KUKA KRL program: Comm010Config.src, Comm010Config.dat

--- Comm010Config.src ---
&ACCESS RVO1
&COMMENT Comm010 Config
&PARAM EDITMASK = *
&PARAM TEMPLATE = C:\KRC\Roboter\Template\vorgabe
&PARAM DISKPATH = KRC:\R1\Program\SbtComm010Stack
DEF Comm010Config( )
;FOLD INI;%{PE}
  ;FOLD BASISTECH INI
    GLOBAL INTERRUPT DECL 3 WHEN $STOPMESS==TRUE DO IR_STOPM ( )
    INTERRUPT ON 3
    BAS (#INITMOV,0 )
  ;ENDFOLD (BASISTECH INI)
  ;FOLD USER INI
    ;Make your modifications here

  ;ENDFOLD (USER INI)
;ENDFOLD (INI)
;FOLD Basic.SetBusCommTimeout IN Timeout: -1 ms ;%{PE}
BusTimeout = -1
;ENDFOLD
;FOLD SbtComm010.FsConfig IN Fs Id: 1, IN Max: Max1, IN Min: Min1 ;%{PE}
Comm010LimUp[1] = Max1
Comm010LimDown[1] = Min1
;ENDFOLD
;FOLD SbtComm010.FsConfig IN Fs Id: 2, IN Max: Max2, IN Min: Min2 ;%{PE}
Comm010LimUp[2] = Max2
Comm010LimDown[2] = Min2
;ENDFOLD
;FOLD SbtComm010.FsConfig IN Fs Id: 3, IN Max: Max3, IN Min: Min3 ;%{PE}
Comm010LimUp[3] = Max3
Comm010LimDown[3] = Min3
;ENDFOLD
;FOLD SbtComm010.FsConfig IN Fs Id: 4, IN Max: Max4, IN Min: Min4 ;%{PE}
Comm010LimUp[4] = Max4
Comm010LimDown[4] = Min4
;ENDFOLD
;FOLD SbtComm010.FsConfig IN Fs Id: 5, IN Max: Max5, IN Min: Min5 ;%{PE}
Comm010LimUp[5] = Max5
Comm010LimDown[5] = Min5
;ENDFOLD
;FOLD SbtComm010.FsConfig IN Fs Id: 6, IN Max: Max6, IN Min: Min6 ;%{PE}
Comm010LimUp[6] = Max6
Comm010LimDown[6] = Min6
;ENDFOLD
;FOLD SbtComm010.FsConfig IN Fs Id: 7, IN Max: Max7, IN Min: Min7 ;%{PE}
Comm010LimUp[7] = Max7
Comm010LimDown[7] = Min7
;ENDFOLD
;FOLD SbtComm010.FsConfig IN Fs Id: 8, IN Max: Max8, IN Min: Min8 ;%{PE}
Comm010LimUp[8] = Max8
Comm010LimDown[8] = Min8
;ENDFOLD


END

--- Comm010Config.dat ---
&ACCESS RVO1
&PARAM EDITMASK = *
&PARAM TEMPLATE = C:\KRC\Roboter\Template\vorgabe
&PARAM DISKPATH = KRC:\R1\Program\SbtComm010Stack
DEFDAT Comm010Config
;FOLD EXTERNAL DECLARATIONS;%{PE}%MKUKATPBASIS,%CEXT,%VCOMMON,%P
;FOLD BASISTECH EXT;%{PE}%MKUKATPBASIS,%CEXT,%VEXT,%P
EXT  BAS (BAS_COMMAND  :IN,REAL  :IN )
DECL INT SUCCESS
;ENDFOLD (BASISTECH EXT)
;FOLD USER EXT;%{E}%MKUKATPUSER,%CEXT,%VEXT,%P
;Make your modifications here

;ENDFOLD (USER EXT)
;ENDFOLD (EXTERNAL DECLARATIONS)
DECL vector_t Max1={X 3000.00,Y 3000.00,Z 3000.00}
DECL vector_t Min1={X -3000.00,Y -3000.00,Z -3000.00}
DECL MODULEPARAM_T LAST_TP_PARAMS={PARAMS[] "SBTCOMM010.FSID=8; SBTCOMM010.MAX=Max8; SBTCOMM010.MIN=Min8; BASIC.TIMEOUT=-1    "}
DECL vector_t Max2={X 3000.00,Y 3000.00,Z 3000.00}
DECL vector_t Min2={X -3000.00,Y -3000.00,Z -3000.00}
DECL vector_t Max3={X 3000.00,Y 3000.00,Z 3000.00}
DECL vector_t Min3={X -3000.00,Y -3000.00,Z -3000.00}
DECL vector_t Max4={X 3000.00,Y 3000.00,Z 3000.00}
DECL vector_t Min4={X -3000.00,Y -3000.00,Z -3000.00}
DECL vector_t Max5={X 3000.00,Y 3000.00,Z 3000.00}
DECL vector_t Min5={X -3000.00,Y -3000.00,Z -3000.00}
DECL vector_t Max6={X 3000.00,Y 3000.00,Z 3000.00}
DECL vector_t Min6={X -3000.00,Y -3000.00,Z -3000.00}
DECL vector_t Max7={X 3000.00,Y 3000.00,Z 3000.00}
DECL vector_t Min7={X -3000.00,Y -3000.00,Z -3000.00}
DECL vector_t Max8={X 3000.00,Y 3000.00,Z 3000.00}
DECL vector_t Min8={X -3000.00,Y -3000.00,Z -3000.00}
ENDDAT
